(* CoDeSys 2.3.9.47 project: ats_l3_1.pro *)
(* Libraries: STANDARD.LIB 5.6.98 11:03:02 *)

(* Task configuration *)
TASK Standard (PRIORITY := 0, INTERVAL := T#10ms);
	MAIN_A1
END_TASK

(* Global variable list: Global_Variables *)
VAR_GLOBAL
	btnY	AT%I*	:BOOL;
	btnB	AT%I*	:BOOL;
	lmpG	AT%Q*	:BOOL;
	lmpR	AT%Q*	:BOOL;
END_VAR

(* Global variable list: TwinCAT_Configuration *)
(* Generated automatically by TwinCAT - (read only) *)
VAR_CONFIG
	.btnY AT %IX0.0 : BOOL;
	.btnB AT %IX0.1 : BOOL;
	.lmpG AT %QX0.0 : BOOL;
	.lmpR AT %QX0.1 : BOOL;
END_VAR

(* Data type *)
TYPE SafeState :
(
	sSt_init,
	sSt_changeCode,
	sSt_close,
	sSt_wrongCode,
	sSt_checkDigit,
	sSt_open
);
END_TYPE

(* Data type *)
TYPE T_STATE :
(
	STATE_IDLE := 0,
	STATE_RISE1:= 1,
	STATE_RISE2:= 2,
	STATE_FALL1:= 3,
	STATE_FALL2:= 4
);
END_TYPE

(* POU MAIN_A1, ST *)
PROGRAM MAIN_A1
VAR
	(*Program used Variables*)
	currentSafeState 	: SafeState;
	codeArray			: ARRAY[1..4] OF BOOL:= FALSE, FALSE, FALSE, FALSE;
	currentIndex		: INT := 1;
	correctCounter		: INT := 0;
	t_abs				: REAL:= 0;
	lightCounter		: INT := 0;
	(*Objects*)
	EdgDect_Y			: DoubleEdgeDetector;
	EdgDect_B			: DoubleEdgeDetector;
	(*EdgeDetector used Variables*)
	t_Y					: REAL := 0; (*Measure Time between two same Edges*)
	t_B					: REAL := 0; (*Measure Time between two same Edges*)
END_VAR
VAR CONSTANT
	lightDuration		: INT := 5; 	(*Seconds*)
	t_blind				: REAL:= 0.2; 	(*Seconds*)
END_VAR
(*Initialize EdgeDetectors*)
EdgDect_Y();
EdgDect_B();

(*Scan Button Y*)
EdgDect_Y.sig_in := btnY;
EdgDect_Y.Ti	 := t_blind;
EdgDect_Y.t		 := t_Y;
(*Scan Button B*)
EdgDect_B.sig_in := btnB;
EdgDect_B.Ti	 := t_blind;
EdgDect_B.t		 := t_B;


(*Final State Machine (FSM)*)
CASE currentSafeState OF


	sSt_init:
		(*Fill Array with secret Code*)
		codeArray[1]:= TRUE;
		codeArray[2]:= FALSE;
		codeArray[3]:= FALSE;
		codeArray[4]:= TRUE;
		(*Branch to State "Close"*)
		currentSafeState := sSt_close;


	sSt_close:
		(*Fuck Everything*)
		currentIndex	:= 1;
		correctCounter	:= 0;
		lmpG			:= FALSE;
		lmpR			:= FALSE;
		lightCounter	:= 100*lightDuration;
		(*Branch to State "Check Digit"*)
		currentSafeState := sSt_checkDigit;

	sSt_changeCode:

		lmpG	:= TRUE;
		lmpR	:= TRUE;

		IF EdgDect_Y.rise = TRUE THEN
			codeArray[currentIndex]:= FALSE;
			currentIndex := currentIndex + 1;
		ELSIF EdgDect_B.rise = TRUE THEN
			codeArray[currentIndex]:= TRUE;
			currentIndex := currentIndex + 1;
		END_IF

		IF currentIndex > 4 THEN
			currentSafeState := sSt_close;
		END_IF
		


	sSt_wrongCode:
		lmpG	:= FALSE;
		lmpR	:= TRUE;
		
		(*Decrement Light Duration Counter*)	
		lightCounter := lightCounter - 1;

		IF lightCounter <= 0 THEN
			currentSafeState := sSt_close;
		END_IF

	sSt_checkDigit:
		(*Just if a Button is pressed...*)
		IF EdgDect_Y.rise = TRUE THEN
			IF codeArray[currentIndex] = FALSE THEN
				correctCounter := correctCounter + 1;
			ELSE
				correctCounter := 0;
			END_IF
			(*Increment for checking next Entry*)
			currentIndex := currentIndex +1;
		ELSIF EdgDect_B.rise = TRUE THEN
			IF codeArray[currentIndex] = TRUE THEN
				correctCounter := correctCounter + 1;
			ELSE
				correctCounter := 0;
			END_IF
			(*Increment for checking next Entry*)
			currentIndex := currentIndex +1;
		END_IF
		
		IF correctCounter = 4 THEN
			(*Branch to State "Open"*)
			currentSafeState := sSt_open;
		ELSIF (currentIndex = 5) AND (correctCounter <> 4) THEN
			(*Branch to State "Wrong Code"*)
			currentSafeState := sSt_wrongCode;
		ELSE
			(*Remain*)
			currentSafeState := sSt_checkDigit;
		END_IF

		IF EdgDect_B.rises = TRUE THEN
			currentSafeState := sSt_close;
		END_IF

	sSt_open:
		lmpG	:= TRUE;
		lmpR	:= FALSE;
			
		(*Branch to change Code if wanted*)
		IF (EdgDect_Y.rise = TRUE) AND (EdgDect_B.rise = TRUE) THEN
			currentIndex := 1;
			currentSafeState := sSt_changeCode;
		END_IF

		(*Decrement Light Duration Counter*)	
		lightCounter := lightCounter - 1;

		IF lightCounter <= 0 THEN
			currentSafeState := sSt_close;
		END_IF

	ELSE
		;
END_CASE;

(*Timer Stuff*)

(*Increment Time t for Button Y*)
IF EdgDect_Y.timer_ON = TRUE THEN
	(*Timer starts counting*)
	t_Y := t_Y + 0.01;
ELSE
	(*Time is up*)
	t_Y := 0;
END_IF

(*Increment Time t for Button B*)
IF EdgDect_B.timer_ON = TRUE THEN
	(*Timer starts counting*)
	t_B := t_B + 0.01;
ELSE
	(*Time is up*)
	t_B := 0;
END_IF

(*Increment Absolute Time*)
t_abs := t_abs + 0.01;
END_PROGRAM

(* POU DoubleEdgeDetector, ST *)
FUNCTION_BLOCK DoubleEdgeDetector
VAR_INPUT
	(*Input Signal*)
	sig_in 		: BOOL ;
	(*Timer Count*)
	t			: REAL ;
	(*Idle Time*)
	Ti			: REAL  ;
END_VAR
VAR_OUTPUT
	fall		: BOOL ;
	falls		: BOOL ;	
	rise		: BOOL ;
	rises		: BOOL ;
	(*Timer Commands*)
	timer_ON	: BOOL ;
END_VAR
VAR
	c_state		: T_STATE := STATE_IDLE;
	prev_sig	: BOOL := FALSE;
	edgeRise	: BOOL := FALSE;
	edgeFall	: BOOL := FALSE;
	TOF			: BOOL := FALSE;
END_VAR
(*Reset Outputs*)
DoubleEdgeDetector.fall		:= FALSE ;
DoubleEdgeDetector.falls	:= FALSE ;
DoubleEdgeDetector.rise		:= FALSE ;
DoubleEdgeDetector.rises	:= FALSE ;

(*Check Timer Overflow*)
IF (t > Ti) THEN
	TOF := TRUE;
ELSE
	TOF := FALSE;
END_IF

(*Check Edge*)
IF (prev_sig = sig_in) THEN
	(*Reset Edge*)
	edgeFall := FALSE;
	edgeRise := FALSE;
ELSIF (prev_sig = TRUE) AND (sig_in = FALSE) THEN
	(*Falling Edge*)
	edgeFall := TRUE;
	edgeRise := FALSE;
ELSIF (prev_sig = FALSE) AND (sig_in = TRUE) THEN
	(*Rising Edge*)
	edgeFall := FALSE;
	edgeRise := TRUE;
END_IF

(*Set current Signal = previous Signal*)
prev_sig := sig_in;

(*Final State Machine Implementation*)
CASE c_state OF
	STATE_IDLE:
		(**)
		IF edgeRise = TRUE THEN
			c_state := STATE_RISE1;
		ELSIF edgeFall = TRUE THEN
			c_state := STATE_FALL1;
		ELSE
			c_state := STATE_IDLE;
		END_IF

	STATE_RISE1:
		(*Start Timer*)
		DoubleEdgeDetector.timer_ON := TRUE;
		(**)
		IF TOF = TRUE THEN
			DoubleEdgeDetector.timer_ON := FALSE;
			DoubleEdgeDetector.rise 	:= TRUE;
			c_state := STATE_IDLE;
		ELSIF edgeRise THEN
			c_state := STATE_RISE2;
		ELSE
			c_state := STATE_RISE1;
		END_IF

	STATE_RISE2:
		(**)
		DoubleEdgeDetector.rises 	:= TRUE;
		c_state := STATE_IDLE;
		
	STATE_FALL1:
		(*Start Timer*)
		DoubleEdgeDetector.timer_ON := TRUE;
		(**)
		IF TOF = TRUE THEN
			DoubleEdgeDetector.timer_ON := FALSE;
			DoubleEdgeDetector.fall 	:= TRUE;
			c_state := STATE_IDLE;
		ELSIF edgeFall THEN
			c_state := STATE_FALL2;
		ELSE
			c_state := STATE_FALL1;
		END_IF

	STATE_FALL2:
		(**)
		DoubleEdgeDetector.falls 	:= TRUE;
		c_state := STATE_IDLE;

	ELSE
		c_state := STATE_IDLE;
END_CASE;
END_FUNCTION_BLOCK
